PROGRAM VCC3
VAR
END_VAR

END_PROGRAM

(* stored: Version 1.1.0.1, ProductVersion 3.1.4022.3
   POU VCC3: Id {814a955a-9b99-41f7-82d7-c96e3db38942}, SpecialFunc None *)
